(* CODESYS project tc3_hbi_datalogger.library
   Company: BeckHoff SG
   DefaultNamespace: Tc3_HBI_DataLogger
   Version: 3.1.3.4
   Placeholder: Tc3_HBI_DataLogger
   Title: Tc3_HBI_DataLogger

Project tree, tasks and I/O mapping:
  libraries: Tc2_Standard, * (Beckhoff Automation GmbH); Tc2_System, * (Beckhoff Automation GmbH); Tc2_Utilities, * (Beckhoff Automation GmbH); Tc3_HBI_System, * (BeckHoff)
  DataLogger/
    DUTs/
      data type _ST_DataLogger
      data type _ST_DataLogger_Status
      data type ST_DataLogger
    ITFs/
      interface I_BaseLogger: P_iLogVerbosity, P_sDirectoryPath, P_sFileName, P_sModule, P_sSubDirPath
    function block FB_BaseLogger [ST]: M_nAddBuffer, M_nAddTail, M_nClear, M_nCyclic, M_nDirectory, M_nGetHead, M_RemoveHead, M_sGetToken, P_iLogVerbosity, P_sDirectoryPath, P_sFileName, P_sModule, P_sSubDirPath
  MessageLogger/
    DUTs/
    ITFs/
      interface I_DataLogger
    function block FB_DataLogger [ST]: M_nLogger
  MotorLogger/
    DUTs/
    ITFs/
      interface I_MotorLogger
    function block FB_MotorLogger [ST]: M_nLogger
  SensorLogger/
    DUTs/
    ITFs/
      interface I_SensorLogger
    function block FB_SensorLogger [ST]: M_nLogger
  Version/
    global variables Global_Version
  Tc3_HBI_DataLogger.tmc
*)

// DataLogger/DUTs/_ST_DataLogger
TYPE _ST_DataLogger EXTENDS Tc3_HBI_System.ST_Basic :
STRUCT
	sLogDescription   : STRING; //Info, Error, Warning, Debug
	sLogTstamp  : STRING;
	sLogSource  : STRING; //Cmd from TA, Event to TA, Send done, 
	sLogContent : STRING(255); //The content
END_STRUCT
END_TYPE

// DataLogger/DUTs/_ST_DataLogger_Status
TYPE _ST_DataLogger_Status EXTENDS Tc3_HBI_System.ST_Basic_Status :
STRUCT
END_STRUCT
END_TYPE

// DataLogger/DUTs/ST_DataLogger
TYPE ST_DataLogger EXTENDS _ST_DataLogger :
STRUCT
	stStatus: _ST_DataLogger;
END_STRUCT
END_TYPE

// Version/Global_Version
{attribute 'TcGenerated'}
// This function has been automatically generated from the project information.
VAR_GLOBAL CONSTANT
	{attribute 'const_non_replaced'}
	{attribute 'linkalways'}
	stLibVersion_Tc3_HBI_DataLogger : ST_LibVersion := (iMajor := 3, iMinor := 1, iBuild := 3, iRevision := 4, sVersion := '3.1.3.4');
END_VAR

// DataLogger/ITFs/I_BaseLogger
INTERFACE I_BaseLogger EXTENDS Tc3_HBI_System.I_Basic

PROPERTY P_iLogVerbosity : INT
GET
END_GET
SET
END_SET
END_PROPERTY

PROPERTY P_sDirectoryPath : T_MaxString
GET
END_GET
SET
END_SET
END_PROPERTY

PROPERTY P_sFileName : T_MaxString
GET
END_GET
SET
END_SET
END_PROPERTY

PROPERTY P_sModule : STRING
GET
END_GET
SET
END_SET
END_PROPERTY

PROPERTY P_sSubDirPath : T_MaxString
GET
END_GET
SET
END_SET
END_PROPERTY

END_INTERFACE

// DataLogger/FB_BaseLogger
FUNCTION_BLOCK PUBLIC FB_BaseLogger EXTENDS FB_Basic IMPLEMENTS I_BaseLogger
VAR_INPUT
	sFileName: STRING(80);	
END_VAR
VAR_OUTPUT
END_VAR
VAR	
	FB_BaseDataLogger_DirectoryPath:	T_MAXSTRING:='C:\';
	FB_BaseDataLogger_SubDirPath:		T_MAXSTRING:='AEM\Data\ControllerLog';
	FB_BaseDataLogger_sFileName:		T_MAXSTRING:='System';	
	
	_localData			: _ST_DataLogger;
	_sLine 				: T_MAXSTRING;
	
	_SysTimeStamp 		: STRING; //format YYYY/MM/dd HH:mm:ss:nnn	
	_systemTime			: TIMESTRUCT;
	fbLocalTime 		: FB_LocalSystemTime;
	fbFormatString		: FB_FormatString;
	sYear				: STRING ;
	sMonth 				: T_MAXSTRING;
	sDay 				: T_MAXSTRING;
	sHour				: T_MAXSTRING;
	sMinute				: T_MAXSTRING;
	sSecond 			: T_MAXSTRING;
	sMiliSec 			: T_MAXSTRING;
	
	fbFileOpen			: FB_FileOpen;
	fbFileClose			: FB_FileClose;
	fbFilePuts			: FB_FilePuts;
	fbCreateDir			: FB_CreateDir;
	fbEnumFindFileEntry	: FB_EnumFindFileEntry;
	
	_SysTimeStamp2		: STRING(255);
	FB_BaseDataLogger_iLogVerbosity 		: INT:= 5;
	FB_BaseDataLogger_M_nCyclic_iState: INT;
	FB_BaseDataLogger_sModule	: STRING(80);
// Queue
	arrBuffer : ARRAY [0..MAX_BUFFER_SIZE] OF _ST_DataLogger;
	fbBuffer : FB_MemRingBuffer;
	nCount : UDINT;
	nLoad: UDINT;
// Directory
	FB_BaseLogger_M_nDirectory_iState	: INT;
	FB_BaseLogger_M_nDirectory_bExecute: BOOL;
	FB_BaseLogger_M_nDirectory_fbExecute: R_TRIG;
	
	FB_BaseLogger_M_nDirectory_sSubDirPath: T_MAXSTRING;
	FB_BaseLogger_M_nDirectory_sSubDirPath1: T_MAXSTRING;
	FB_BaseLogger_M_nDirectory_sSubDirPath2: T_MAXSTRING;
	FB_BaseLogger_M_nDirectory_sSubDirPath3: T_MAXSTRING;
	FB_BaseLogger_M_nDirectory_sSubDirPath4: T_MAXSTRING;
	FB_BaseLogger_M_nDirectory_nToken	   : INT;	
END_VAR
VAR CONSTANT
	//Log verbosity
	LOG_LEVEL_ERROR   	: INT := 5;
	LOG_LEVEL_WARNING 	: INT := 4;
	LOG_LEVEL_MESSAGE 	: INT := 3;
	LOG_LEVEL_INFO    	: INT := 2;
	LOG_LEVEL_DEBUG   	: INT := 1;
	MAX_BUFFER_SIZE		: UDINT:= 10000;
END_VAR

METHOD PUBLIC M_nAddBuffer : UDINT
VAR_INPUT
	sLogDescription    : T_MAXSTRING;
	sLogSource         : T_MAXSTRING;
	sLogContent        : T_MAXSTRING;
END_VAR
VAR_IN_OUT
	_localData	   : _ST_DataLogger;
END_VAR
VAR
	fbFormatString : FB_FormatString;
	stLocal: _ST_DataLogger;
END_VAR
IF NOT fbLocalTime.bValid THEN RETURN; END_IF

fbFormatString(sFormat:= '%-7s', arg1:= F_STRING(sLogDescription), sOut => stLocal.sLogDescription);
fbFormatString(sFormat:= '%-15s', arg1:= F_STRING(sLogSource), sOut => stLocal.sLogSource);

stLocal.sLogContent:= sLogContent;
stLocal.sLogTstamp:= _SysTimeStamp;

IF M_nAddTail(stLocal)=Tc3_HBI_System.cCOMPLETE THEN
	M_nAddBuffer:= Tc3_HBI_System.cCOMPLETE;
ELSE
	M_nAddBuffer := Tc3_HBI_System.cPOINTER_OR_INDEX_ERROR;
END_IF
END_METHOD

METHOD PUBLIC M_nAddTail : UDINT
VAR_INPUT
	stAdd : _ST_DataLogger;
END_VAR
fbBuffer.A_AddTail(
	pWrite:= ADR(stAdd), 
	cbWrite:= SIZEOF(stAdd), 
	pBuffer:= ADR(arrBuffer), 
	cbBuffer:= SIZEOF(arrBuffer), 
	bOk=> , 
	nCount=> nCount, 
	cbSize=> , 
	cbReturn=> );
	
IF fbBuffer.bOk THEN
	M_nAddTail:= Tc3_HBI_System.cCOMPLETE;
ELSE
	M_nError(nErrorID:= Tc3_HBI_System.cPOINTER_OR_INDEX_ERROR);
	M_nAddTail:= Tc3_HBI_System.cPOINTER_OR_INDEX_ERROR;
END_IF
END_METHOD

METHOD PUBLIC M_nClear : UDINT
VAR_INPUT
END_VAR
MEMSET( ADR( arrBuffer ), 0, SIZEOF( arrBuffer ) ); (* reset (optional) internal buffer *)

fbBuffer.A_Reset( bOk=> ,nCount => nCount );

nLoad := (fbBuffer.cbSize * 100) / MAX_BUFFER_SIZE;

IF fbBuffer.bOk THEN
	M_nClear:= Tc3_HBI_System.cCOMPLETE;
	ELSE 
		M_nError(nErrorID:= Tc3_HBI_System.cPOINTER_OR_INDEX_ERROR);
		M_nClear:= Tc3_HBI_System.cPOINTER_OR_INDEX_ERROR;
END_IF
END_METHOD

METHOD PUBLIC M_nCyclic : UDINT
VAR_INPUT
END_VAR
//Get current system
	fbLocalTime(
		sNetID:= , 
		bEnable:= TRUE, 
		dwCycle:= , 
		dwOpt:= , 
		tTimeout:= , 
		bValid=> , 
		systemTime=> _systemTime, 
		tzID=> );
		
	sYear 		:= WORD_TO_STRING(_systemtime.wYear);
	sMonth 		:= WORD_TO_STRING(_systemTime.wMonth);
	sDay 		:= WORD_TO_STRING(_systemTime.wDay);
	sHour		:= WORD_TO_STRING(_systemTime.wHour);
	sMinute 	:= WORD_TO_STRING(_systemTime.wMinute);
	sSecond		:= WORD_TO_STRING(_systemTime.wSecond);
	sMilisec 	:= WORD_TO_STRING(_systemTime.wMilliseconds);
		
	fbFormatString(
		sFormat:= '%04s/%02s/%02s %02s:%02s:%02s:%03s', 
		arg1:= F_STRING(sYear), 
		arg2:= F_STRING(sMonth), 
		arg3:= F_STRING(sDay), 
		arg4:= F_STRING(sHour), 
		arg5:= F_STRING(sMinute), 
		arg6:= F_STRING(sSecond), 
		arg7:= F_STRING(sMilisec),
		bError=> , 
		nErrId=> , 
		sOut=> _SysTimeStamp);
		
	fbFormatString(
		sFormat:= '%04s-%02s-%02sT%02s', 
		arg1:= F_STRING(sYear), 
		arg2:= F_STRING(sMonth), 
		arg3:= F_STRING(sDay), 
		arg4:= F_STRING(sHour),
		bError=> , 
		nErrId=> , 
		sOut=> _SysTimeStamp2);
		
	IF _bReset THEN
		IF _bError THEN
			FB_BaseDataLogger_M_nCyclic_iState:= 0;
		END_IF
	END_IF
	
	
// Local variables
	FB_BaseDataLogger_sFileName:= sFileName;
//Write to file
CASE FB_BaseDataLogger_M_nCyclic_iState OF
	
	0: // Init
		fbEnumFindFileEntry(sNetId:= '', bExecute:= FALSE, );
		fbCreateDir(sNetId:= '', bExecute:= FALSE, );
		fbFileOpen(sNetId:= '', bExecute:= FALSE, );
		fbFilePuts(sNetId:= '', bExecute:= FALSE, );
		fbFileClose(sNetId:= '', bExecute:= FALSE, );
		FB_BaseDataLogger_M_nCyclic_iState:= 30;
		
	10: // Check if directory exit
		fbEnumFindFileEntry(
			sNetId:= '', 
			sPathName:= CONCAT(FB_BaseDataLogger_DirectoryPath,FB_BaseDataLogger_SubDirPath), 
			eCmd:= eEnumCmd_First, 
			bExecute:= TRUE, 
			tTimeout:= T#5S, 
			bBusy=> , 
			bError=> , 
			nErrID=> , 
			bEOE=> , 
			stFindFile=> );
		IF NOT fbEnumFindFileEntry.bBusy THEN	
			IF fbEnumFindFileEntry.bError THEN
				M_nError(nErrorID:= fbEnumFindFileEntry.nErrId);
				FB_BaseDataLogger_M_nCyclic_iState:= 999;
			ELSE
				IF NOT fbEnumFindFileEntry.bEOE THEN
					FB_BaseDataLogger_M_nCyclic_iState:= 30; (*target dir is exist*)
					ELSE FB_BaseDataLogger_M_nCyclic_iState:= 20;	(*target dir no exist*)
				END_IF
			END_IF
			fbEnumFindFileEntry(sNetId:= '', bExecute:= FALSE, );
		END_IF
		
	20: // Create directory
		fbCreateDir(
			sNetId:= '', 
			sPathName:= CONCAT(FB_BaseDataLogger_DirectoryPath,FB_BaseDataLogger_SubDirPath), 
			ePath:= PATH_GENERIC, 
			bExecute:= TRUE, 
			tTimeout:= T#5S, 
			bBusy=> , 
			bError=> , 
			nErrId=> );
		IF NOT fbCreateDir.bBusy THEN	
			IF fbCreateDir.bError THEN
				M_nError(nErrorID:= fbCreateDir.nErrId);
				FB_BaseDataLogger_M_nCyclic_iState:= 999;
			ELSE
				FB_BaseDataLogger_M_nCyclic_iState:= 30;	
			END_IF
			fbCreateDir(sNetId:= '', bExecute:= FALSE, );
		END_IF	
	
	30: // Waiting
		IF nCount > 0 THEN
			FB_BaseDataLogger_M_nCyclic_iState := 40;
		END_IF
	
	40: // Open file
		fbFileOpen(
			sNetId:= , 
			sPathName:= CONCAT(CONCAT(FB_BaseDataLogger_DirectoryPath,CONCAT(CONCAT(FB_BaseDataLogger_SubDirPath,'\'),
						CONCAT(FB_BaseDataLogger_sFileName, _SysTimeStamp2))), '.log'),  
			nMode:= FOPEN_MODEAPPEND, 
			ePath:= , 
			bExecute:= TRUE, 
			tTimeout:= , 
			bBusy=> , 
			bError=> , 
			nErrId=> , 
			hFile=> );
		
		IF NOT fbFileOpen.bBusy THEN
			fbFileOpen(bExecute := FALSE);
			IF NOT fbFileOpen.bError THEN
				_localData := M_RemoveHead();
				FB_BaseDataLogger_M_nCyclic_iState := 50;
			ELSE
				M_nError(nErrorID:= fbFileOpen.nErrId);
				FB_BaseDataLogger_M_nCyclic_iState := 999;
			END_IF
		END_IF
	
	50: // Put file
		fbFormatString(
			sFormat:= '"%s" "%s" "%s" "%s"$R$N', 
			arg1:= F_STRING(_localData.sLogTstamp), 
			arg2:= F_STRING(_localData.sLogDescription), 
			arg3:= F_STRING(_localData.sLogSource), 
			arg4:= F_STRING(_localData.sLogContent), 
			sOut=> _sLine);
		
		fbFilePuts(
			sNetId:= , 
			hFile:= fbFileOpen.hFile, 
			sLine:= _sLine, 
			bExecute:= TRUE, 
			tTimeout:= , 
			bBusy=> , 
			bError=> , 
			nErrId=> );
			
		IF NOT fbFilePuts.bBusy THEN
			fbFilePuts(bExecute := FALSE);
			IF NOT fbFilePuts.bError THEN
				IF nCount > 0 THEN //still have data
					_localData := M_RemoveHead();
					FB_BaseDataLogger_M_nCyclic_iState := 50;
				ELSE
					FB_BaseDataLogger_M_nCyclic_iState := 60;
				END_IF
			ELSE
				M_nError(nErrorID:= fbFilePuts.nErrId);
				FB_BaseDataLogger_M_nCyclic_iState := 999;
			END_IF
		END_IF
	
	60: // Close file
		fbFileClose(
			sNetId:= , 
			hFile:= fbFileOpen.hFile, 
			bExecute:= TRUE, 
			tTimeout:= , 
			bBusy=> , 
			bError=> , 
			nErrId=> );
	
		IF NOT fbFileClose.bBusy THEN
			fbFileClose(bExecute := FALSE);
			IF NOT fbFileClose.bError THEN
				FB_BaseDataLogger_M_nCyclic_iState := 70;
			ELSE
				M_nError(nErrorID:= fbFileClose.nErrId);
				FB_BaseDataLogger_M_nCyclic_iState := 999;
			END_IF
		END_IF
	
	70: // Next cycle
		IF nCount > 0 THEN
			FB_BaseDataLogger_M_nCyclic_iState := 30;
		END_IF
	999: // Error state
		fbEnumFindFileEntry(sNetId:= '', bExecute:= FALSE, );
		fbCreateDir(sNetId:= '', bExecute:= FALSE, );
		fbFileOpen(sNetId:= '', bExecute:= FALSE, );
		fbFilePuts(sNetId:= '', bExecute:= FALSE, );
		fbFileClose(sNetId:= '', bExecute:= FALSE, );
		
	ELSE FB_BaseDataLogger_M_nCyclic_iState:= 0;
	
END_CASE
END_METHOD

METHOD PUBLIC M_nDirectory : UDINT
VAR_INPUT
	bExecute: BOOL;
END_VAR
VAR	
END_VAR
FB_BaseLogger_M_nDirectory_bExecute:= bExecute;
FB_BaseLogger_M_nDirectory_fbExecute(CLK:= FB_BaseLogger_M_nDirectory_bExecute, Q=> );

IF FB_BaseLogger_M_nDirectory_fbExecute.Q THEN
	FB_BaseLogger_M_nDirectory_iState:= 10;
END_IF

	FB_BaseLogger_M_nDirectory_sSubDirPath1:= M_sGetToken(sAllTokens:= FB_BaseDataLogger_SubDirPath, nToken:= 1, sDelim:= '\');
	FB_BaseLogger_M_nDirectory_sSubDirPath2:= M_sGetToken(sAllTokens:= FB_BaseDataLogger_SubDirPath, nToken:= 2, sDelim:= '\');
	FB_BaseLogger_M_nDirectory_sSubDirPath3:= M_sGetToken(sAllTokens:= FB_BaseDataLogger_SubDirPath, nToken:= 3, sDelim:= '\');
	FB_BaseLogger_M_nDirectory_sSubDirPath4:= M_sGetToken(sAllTokens:= FB_BaseDataLogger_SubDirPath, nToken:= 4, sDelim:= '\');
	
	IF FB_BaseLogger_M_nDirectory_sSubDirPath1='' OR FB_BaseLogger_M_nDirectory_sSubDirPath4<> '' THEN
		M_nError(nErrorID:= Tc3_HBI_System.cPARAMETER_ERROR);
		M_nDirectory:= Tc3_HBI_System.cPARAMETER_ERROR;
		RETURN;
	END_IF
	
IF _bReset THEN
	IF _bError THEN
		FB_BaseLogger_M_nDirectory_iState:= 0;
	END_IF
END_IF

CASE FB_BaseLogger_M_nDirectory_iState OF
 
	0: // Init
		M_nDirectory:= Tc3_HBI_System.cIDLE;
		
		fbEnumFindFileEntry(sNetId:= '', bExecute:= FALSE, );
		fbCreateDir(sNetId:= '', bExecute:= FALSE, );
		
	10: // Check if directory exit
		M_nDirectory:= Tc3_HBI_System.cRUNNING;
		
		fbEnumFindFileEntry(
			sNetId:= '', 
			sPathName:= CONCAT(FB_BaseDataLogger_DirectoryPath,FB_BaseDataLogger_SubDirPath), 
			eCmd:= eEnumCmd_First, 
			bExecute:= TRUE, 
			tTimeout:= T#5S, 
			bBusy=> , 
			bError=> , 
			nErrID=> , 
			bEOE=> , 
			stFindFile=> );
		IF NOT fbEnumFindFileEntry.bBusy THEN	
			IF fbEnumFindFileEntry.bError THEN
				M_nError(nErrorID:= fbEnumFindFileEntry.nErrId);
				FB_BaseLogger_M_nDirectory_iState:= 999;
			ELSE
				IF NOT fbEnumFindFileEntry.bEOE THEN
					FB_BaseLogger_M_nDirectory_iState:= 70; (*target dir is exist*)
					ELSE 
						FB_BaseLogger_M_nDirectory_sSubDirPath:= FB_BaseLogger_M_nDirectory_sSubDirPath1;
						FB_BaseLogger_M_nDirectory_iState:= 20;	(*target dir no exist*)
				END_IF
			END_IF
			fbEnumFindFileEntry(sNetId:= '', bExecute:= FALSE, );
		END_IF	
		
	20: // Create directory
		M_nDirectory:= Tc3_HBI_System.cRUNNING;
		
		fbCreateDir(
			sNetId:= '', 
			sPathName:= CONCAT(FB_BaseDataLogger_DirectoryPath,FB_BaseLogger_M_nDirectory_sSubDirPath), 
			ePath:= PATH_GENERIC, 
			bExecute:= TRUE, 
			tTimeout:= T#5S, 
			bBusy=> , 
			bError=> , 
			nErrId=> );
		IF NOT fbCreateDir.bBusy THEN	
			IF fbCreateDir.bError THEN
				M_nError(nErrorID:= fbCreateDir.nErrId);
				FB_BaseLogger_M_nDirectory_iState:= 999;
			ELSE
				FB_BaseLogger_M_nDirectory_iState:= 30;	
			END_IF
			fbCreateDir(sNetId:= '', bExecute:= FALSE, );
		END_IF
		
	30: // Create directory
		M_nDirectory:= Tc3_HBI_System.cRUNNING;
		
		IF FB_BaseLogger_M_nDirectory_sSubDirPath1<> FB_BaseLogger_M_nDirectory_sSubDirPath2 THEN
			FB_BaseLogger_M_nDirectory_sSubDirPath:= CONCAT(FB_BaseLogger_M_nDirectory_sSubDirPath1,CONCAT('\',FB_BaseLogger_M_nDirectory_sSubDirPath2));
			FB_BaseLogger_M_nDirectory_iState:= 40;
			ELSE FB_BaseLogger_M_nDirectory_iState:= 70;
		END_IF
		
 	40: // Create directory
		M_nDirectory:= Tc3_HBI_System.cRUNNING;
		
		fbCreateDir(
			sNetId:= '', 
			sPathName:= CONCAT(FB_BaseDataLogger_DirectoryPath,FB_BaseLogger_M_nDirectory_sSubDirPath), 
			ePath:= PATH_GENERIC, 
			bExecute:= TRUE, 
			tTimeout:= T#5S, 
			bBusy=> , 
			bError=> , 
			nErrId=> );
		IF NOT fbCreateDir.bBusy THEN	
			IF fbCreateDir.bError THEN
				M_nError(nErrorID:= fbCreateDir.nErrId);
				FB_BaseLogger_M_nDirectory_iState:= 999;
			ELSE
				FB_BaseLogger_M_nDirectory_iState:= 50;	
			END_IF
			fbCreateDir(sNetId:= '', bExecute:= FALSE, );
		END_IF
		
	50: // Create directory
		M_nDirectory:= Tc3_HBI_System.cRUNNING;
		
		IF FB_BaseLogger_M_nDirectory_sSubDirPath2<> FB_BaseLogger_M_nDirectory_sSubDirPath3 THEN
			FB_BaseLogger_M_nDirectory_sSubDirPath:= CONCAT(CONCAT(FB_BaseLogger_M_nDirectory_sSubDirPath1,'\'),
							CONCAT(FB_BaseLogger_M_nDirectory_sSubDirPath2,CONCAT('\',FB_BaseLogger_M_nDirectory_sSubDirPath3)));
			FB_BaseLogger_M_nDirectory_iState:= 60;
			ELSE FB_BaseLogger_M_nDirectory_iState:= 70;
		END_IF
		
	60: // Create directory
		M_nDirectory:= Tc3_HBI_System.cRUNNING;
		
		fbCreateDir(
			sNetId:= '', 
			sPathName:= CONCAT(FB_BaseDataLogger_DirectoryPath,FB_BaseLogger_M_nDirectory_sSubDirPath), 
			ePath:= PATH_GENERIC, 
			bExecute:= TRUE, 
			tTimeout:= T#5S, 
			bBusy=> , 
			bError=> , 
			nErrId=> );
		IF NOT fbCreateDir.bBusy THEN	
			IF fbCreateDir.bError THEN
				M_nError(nErrorID:= fbCreateDir.nErrId);
				FB_BaseLogger_M_nDirectory_iState:= 999;
			ELSE
				FB_BaseLogger_M_nDirectory_iState:= 70;	
			END_IF
			fbCreateDir(sNetId:= '', bExecute:= FALSE, );
		END_IF

	70: // Done
		M_nDirectory:= Tc3_HBI_System.cCOMPLETE;
		IF NOT FB_BaseLogger_M_nDirectory_bExecute THEN
			FB_BaseLogger_M_nDirectory_bExecute:= 0;
		END_IF
	
	999: // Error state
		;
	
	ELSE FB_BaseLogger_M_nDirectory_iState:= 0;
		
END_CASE
END_METHOD

METHOD PUBLIC M_nGetHead : UDINT
VAR_INPUT
END_VAR
fbBuffer.A_GetHead( pRead:= ADR( M_nGetHead ),
					cbRead:= SIZEOF( M_nGetHead ),
					pBuffer:= ADR( arrBuffer ),
					cbBuffer:= SIZEOF( arrBuffer ),
					bOk=> ,
					nCount => nCount );

nLoad := (fbBuffer.cbSize * 100) / MAX_BUFFER_SIZE;
END_METHOD

METHOD PUBLIC M_RemoveHead : _ST_DataLogger
VAR_INPUT
END_VAR
fbBuffer.A_RemoveHead( 	pRead:= ADR( M_RemoveHead ),
						cbRead:= SIZEOF( M_RemoveHead ),
						pBuffer:= ADR( arrBuffer ),
						cbBuffer:= SIZEOF( arrBuffer ),
						bOk=> ,
						nCount => nCount );

nLoad := (fbBuffer.cbSize * 100) / MAX_BUFFER_SIZE;
END_METHOD

METHOD PRIVATE M_sGetToken : STRING
VAR_INPUT
	sAllTokens: Tc2_System.T_MaxString;
	nToken: UINT;
  	sDelim: STRING;
END_VAR
VAR
// Temporary Variables 
	pString: POINTER TO STRING;
	nCurTokenLocation: INT;
END_VAR
pString:= ADR(sAllTokens);

IF nToken < 1 OR LEN(sDelim) < 1 THEN
	// Negative OR zeroth token OR empty delimiter strings mean an empty token 
	M_sGetToken:= '';
 	RETURN;
ELSE
	IF nToken = 1 THEN
	// Quickly extract the first token 
	nCurTokenLocation:= FIND(pString^, sDelim);
	   	IF nCurTokenLocation > 1 THEN
	   		M_sGetToken:= LEFT(pString^, nCurTokenLocation - 1);
	   	ELSE
			M_sGetToken:= pString^;
	    END_IF
	ELSE
		// FIND the Nth token 
		REPEAT
			nCurTokenLocation:= FIND(pString^, sDelim);
			IF nCurTokenLocation = 0 THEN
				M_sGetToken:= '';
				RETURN;
			ELSE
				pString:= pString + INT_TO_DWORD(nCurTokenLocation -1) + INT_TO_DWORD(LEN(sDelim));
			END_IF
	
			nToken:= nToken - 1;
			UNTIL nToken = 1
		END_REPEAT;

		// Extract the Nth token (Which is the next token AT this point) 
		nCurTokenLocation:= FIND(pString^, sDelim);
		IF nCurTokenLocation > 0 THEN
			M_sGetToken:= LEFT(pString^, nCurTokenLocation - 1);
			RETURN;
		ELSE
			M_sGetToken:= pString^;
		   	RETURN;
		END_IF
	END_IF
END_IF
END_METHOD

PROPERTY PUBLIC P_iLogVerbosity : INT
GET
P_iLogVerbosity := FB_BaseDataLogger_iLogVerbosity;
END_GET
SET
IF P_iLogVerbosity< 1 THEN
	FB_BaseDataLogger_iLogVerbosity:= 1;
ELSE 
	IF P_iLogVerbosity> 5 THEN
		P_iLogVerbosity:= 5;
	ELSE FB_BaseDataLogger_iLogVerbosity := P_iLogVerbosity;		
	END_IF
END_IF
END_SET
END_PROPERTY

PROPERTY PUBLIC P_sDirectoryPath : T_MaxString
GET
P_sDirectoryPath:= FB_BaseDataLogger_DirectoryPath;
END_GET
SET
FB_BaseDataLogger_DirectoryPath:= P_sDirectoryPath;
END_SET
END_PROPERTY

PROPERTY P_sFileName : T_MaxString
GET
P_sFileName:= FB_BaseDataLogger_sFileName;
END_GET
SET
FB_BaseDataLogger_sFileName:= P_sFileName;
END_SET
END_PROPERTY

PROPERTY P_sModule : STRING
GET
P_sModule:= FB_BaseDataLogger_sModule;
END_GET
SET
FB_BaseDataLogger_sModule:= P_sModule;
END_SET
END_PROPERTY

PROPERTY PUBLIC P_sSubDirPath : T_MaxString
GET
P_sSubDirPath:= FB_BaseDataLogger_SubDirPath;
END_GET
SET
FB_BaseDataLogger_SubDirPath:= P_sSubDirPath;
END_SET
END_PROPERTY

END_FUNCTION_BLOCK

// MessageLogger/ITFs/I_DataLogger
INTERFACE I_DataLogger EXTENDS I_BaseLogger

END_INTERFACE

// MessageLogger/FB_DataLogger
FUNCTION_BLOCK PUBLIC FB_DataLogger EXTENDS FB_BaseLogger IMPLEMENTS I_DataLogger
VAR_INPUT
END_VAR
VAR_OUTPUT
END_VAR
VAR
	FB_DataLogger_M_nLogger_iLogLevel: INT:= 5;
	FB_DataLogger_M_nLogger_sSource: STRING(80);
	FB_DataLogger_M_nLogger_sMessage: STRING(255);
END_VAR

METHOD PUBLIC M_nLogger : UDINT
VAR_INPUT
	iLogLevel	: INT:= 5;
	sSource : STRING(80);
	sMessage: STRING(255);
END_VAR
FB_DataLogger_M_nLogger_iLogLevel:= iLogLevel;

IF FB_DataLogger_M_nLogger_iLogLevel< 1 THEN
	FB_DataLogger_M_nLogger_iLogLevel:= 1;
	ELSE
		IF FB_DataLogger_M_nLogger_iLogLevel> 5 THEN
 			FB_DataLogger_M_nLogger_iLogLevel:= 5;
		ELSE FB_DataLogger_M_nLogger_iLogLevel:= iLogLevel;
		END_IF
END_IF

IF FB_DataLogger_M_nLogger_iLogLevel > FB_BaseDataLogger_iLogVerbosity THEN
	RETURN; 
END_IF

IF FB_DataLogger_M_nLogger_sSource<> sSource THEN
	M_nAddBuffer(FB_BaseDataLogger_sModule, sSource, sMessage, _localData);
	FB_DataLogger_M_nLogger_sSource:= sSource;
	FB_DataLogger_M_nLogger_sMessage:= sMessage;
ELSE
	IF FB_DataLogger_M_nLogger_sMessage<> sMessage THEN
		M_nAddBuffer(FB_BaseDataLogger_sModule, sSource, sMessage, _localData);
		FB_DataLogger_M_nLogger_sMessage:= sMessage;
		FB_DataLogger_M_nLogger_sSource:= sSource;
	END_IF
END_IF

M_nLogger:= Tc3_HBI_System.cCOMPLETE;
END_METHOD

END_FUNCTION_BLOCK

// MotorLogger/ITFs/I_MotorLogger
INTERFACE I_MotorLogger EXTENDS I_DataLogger

END_INTERFACE

// MotorLogger/FB_MotorLogger
FUNCTION_BLOCK PUBLIC FB_MotorLogger EXTENDS FB_BaseLogger IMPLEMENTS I_MotorLogger
VAR_INPUT
END_VAR
VAR_OUTPUT
END_VAR
VAR
	FB_MotorLogger_M_nLogger_iLogLevel: INT:= 5;
	FB_MotorLogger_M_nLogger_uErrorID: UDINT;
END_VAR

METHOD PUBLIC M_nLogger : UDINT
VAR_INPUT
	iLogLevel	: INT:= 5;
	sMotorName: STRING;
	uErrorID: UDINT;
END_VAR
(*
IF (FB_MotorLogger_M_nLogger_bError <> bError) THEN
	fbFormatString(
		sFormat:= '[%8s %d] : %d', 
		arg1:= F_STRING(FB_BaseLogger_sModule), 
		arg2:= F_INT(iMotorNo), 
		arg3:= F_UDINT(uErrorID),  
		bError=> , 
		nErrId=> , 
		sOut=> );
		
	M_nAddBuffer(FB_BaseLogger_sDescription, 
               CONCAT(CONCAT(BOOL_TO_STRING(FB_MotorLogger_M_nLogger_bError), '->'), BOOL_TO_STRING(bError)), 
               fbFormatString.sOut, _localData);
	FB_MotorLogger_M_nLogger_bError := bError;
END_IF

M_nLogger:= Tc3_HBI_System.cCOMPLETE;
*)

// New
FB_MotorLogger_M_nLogger_iLogLevel:= iLogLevel;

IF FB_MotorLogger_M_nLogger_iLogLevel< 1 THEN
	FB_MotorLogger_M_nLogger_iLogLevel:= 1;
	ELSE
		IF FB_MotorLogger_M_nLogger_iLogLevel> 5 THEN
 			FB_MotorLogger_M_nLogger_iLogLevel:= 5;
		ELSE FB_MotorLogger_M_nLogger_iLogLevel:= iLogLevel;
		END_IF
END_IF

IF FB_MotorLogger_M_nLogger_iLogLevel > FB_BaseDataLogger_iLogVerbosity THEN
	RETURN; 
END_IF

IF (FB_MotorLogger_M_nLogger_uErrorID<> uErrorID) THEN
	
	M_nAddBuffer(FB_BaseDataLogger_sModule, CONCAT(sMotorName,'->'), UDINT_TO_STRING(uErrorID), _localData);
	
	FB_MotorLogger_M_nLogger_uErrorID := uErrorID;
	
END_IF

M_nLogger:= Tc3_HBI_System.cCOMPLETE;
END_METHOD

END_FUNCTION_BLOCK

// SensorLogger/ITFs/I_SensorLogger
INTERFACE I_SensorLogger EXTENDS I_DataLogger

END_INTERFACE

// SensorLogger/FB_SensorLogger
FUNCTION_BLOCK PUBLIC FB_SensorLogger EXTENDS FB_BaseLogger IMPLEMENTS I_SensorLogger
VAR_INPUT
END_VAR
VAR_OUTPUT
END_VAR
VAR
	FB_SensorLogger_M_nLogger_iLogLevel: INT:= 5;
	FB_SensorLogger_M_nLogger_bSensor : BOOL;
END_VAR

METHOD PUBLIC M_nLogger : UDINT
VAR_INPUT
	iLogLevel	: INT:= 5;
	sSensorName : STRING;
	bSensor  : BOOL;
END_VAR
FB_SensorLogger_M_nLogger_iLogLevel:= iLogLevel;

IF FB_SensorLogger_M_nLogger_iLogLevel< 1 THEN
	FB_SensorLogger_M_nLogger_iLogLevel:= 1;
	ELSE
		IF FB_SensorLogger_M_nLogger_iLogLevel> 5 THEN
 			FB_SensorLogger_M_nLogger_iLogLevel:= 5;
		ELSE FB_SensorLogger_M_nLogger_iLogLevel:= iLogLevel;
		END_IF
END_IF

IF FB_SensorLogger_M_nLogger_iLogLevel > FB_BaseDataLogger_iLogVerbosity THEN
	RETURN; 
END_IF

IF (FB_SensorLogger_M_nLogger_bSensor <> bSensor) THEN
	M_nAddBuffer(FB_BaseDataLogger_sModule, 
               CONCAT(CONCAT(BOOL_TO_STRING(FB_SensorLogger_M_nLogger_bSensor),'->'),BOOL_TO_STRING(bSensor)), 
               sSensorName, _localData);
	FB_SensorLogger_M_nLogger_bSensor := bSensor;
END_IF

M_nLogger:= Tc3_HBI_System.cCOMPLETE;
END_METHOD

END_FUNCTION_BLOCK
